Staubli VAL3: getCaption.pgx

public program getCaption(string& x_sCaption[])
// This program returns le caption of the textboxes
  local num l_i
begin
  l_i=0
  while (l_i<nNumOfTxtBox)
    if l_i<size(x_sCaption)
      x_sCaption[l_i]=pw:sTxtBoxCaption[l_i]
    endIf
    l_i=l_i+1
  endWhile
end
